TYPE AX52XXDriveChannelStatuses :
STRUCT
	///Is the drive in a busy state?
	busyStatus: BusyStatus;
	///Is the drive in a healthy state?
	healthStatus: HealthStatus;
END_STRUCT
END_TYPE

(* stored: Version 1.1.0.1, ProductVersion 3.1.4019.2
   DUT AX52XXDriveChannelStatuses: Id {7a170891-647b-4b73-ae09-1f13727e578e} *)
